FUNCTION_BLOCK FB_Valve
VAR_INPUT
END_VAR
VAR_OUTPUT
END_VAR
VAR
	Value 		: LREAL;
	Parameters 	: ST_ValveParam := (Set := 1, P := 2, I := 3, D := 4, Unit:='Deg');
END_VAR

Value := HMI.SineVerySlow*180/2;

END_FUNCTION_BLOCK

(* stored: Version 1.1.0.1, ProductVersion 3.1.4022.18
   POU FB_Valve: Id {7e198f3d-5c76-4053-b222-a991847d3cc2}, SpecialFunc None *)
